{attribute 'qualified_only'}
{attribute 'strict'}
TYPE BoxStatus :
(
	enum_member := 0
);
END_TYPE

(* stored: Version 1.1.0.1, ProductVersion 3.1.4024.13
   DUT BoxStatus: Id {f7c1fa11-7adb-468b-8fd2-ae68f47f1d98} *)
